# B&R Automation Studio project Lib1Lab1
Automation Studio 4.5.2.102

## Configuration Config1

CPU 4PP065.0571-P74, AutomationRuntime D4.52, Build 4.1.2, Vc V4.52.0

### Task classes (Cpu.sw)
```
Cyclic#1:
  Program <- Program.prg
Binaries: udbdef, TCData, ashwd, User, asfw, arconfig, sysconf, Role, ashwac, iomap
Libraries: LOR
```

### Hardware
```
4PP065_0571_P74 : 4PP065.0571-P74 v1.1.2.0
  Connector IF4:
    SubnetMask = 255.255.255.0
    InaNodeNumber = 1
  Connector IF5:
    ActivateDevice = 1
    Mode = Manual
    InternetAddress = 10.0.1.10
    SubnetMask = 255.255.255.0
  ConfigurationID = labBR
```

## Logical view

Binary libraries used (declarations not repeated): operator, runtime, astime, AsIecCon

### Package Logical/Libraries - Global libraries

### Library Logical/Libraries/LOR (ANSIC)

#### LOR.fun
```iecst
{REDUND_ERROR} FUNCTION_BLOCK FB_Integrator (*TODO: Add your comment here*) (*$GROUP=User,$CAT=User,$GROUPICON=User.png,$CATICON=User.png*)
	VAR_INPUT
		in : REAL;
	END_VAR
	VAR_OUTPUT
		out : REAL;
	END_VAR
	VAR
		dt : REAL;
	END_VAR
END_FUNCTION_BLOCK

{REDUND_ERROR} FUNCTION_BLOCK FB_Motor (*TODO: Add your comment here*) (*$GROUP=User,$CAT=User,$GROUPICON=User.png,$CATICON=User.png*)
	VAR_INPUT
		u : REAL;
	END_VAR
	VAR_OUTPUT
		phi : REAL;
		w : REAL;
	END_VAR
	VAR
		integrator : FB_Integrator;
		Tm : REAL;
		ke : REAL;
		dt : REAL;
	END_VAR
END_FUNCTION_BLOCK

{REDUND_ERROR} FUNCTION_BLOCK FB_Regulator (*TODO: Add your comment here*) (*$GROUP=User,$CAT=User,$GROUPICON=User.png,$CATICON=User.png*)
	VAR_INPUT
		e : REAL; (*рассогласование между задающим воздействием и реальной скоростью вращения вала ДПТ об/мин*)
	END_VAR
	VAR_OUTPUT
		u : REAL; (*напряжение на выходе ДПТ В*)
	END_VAR
	VAR
		k_p : REAL; (*П коэф регулятора*)
		k_i : REAL; (*И коэф регулятора*)
		integrator : FB_Integrator; (*Интегратор*)
		iyOld : REAL; (*храниение предыдущего значения схемы противонакопления*)
		max_abs_value : REAL; (*Umax*)
		dt : REAL; (*хе-хе-хе*)
		e_kp : REAL; (*промежуточное значение вычесления*)
	END_VAR
END_FUNCTION_BLOCK
```

#### FB_Integrator.c
```c
#include <bur/plctypes.h>
#ifdef __cplusplus
	extern "C"
	{
#endif
	#include "LOR.h"
#ifdef __cplusplus
	};
#endif
/* TODO: Add your comment here */
void FB_Integrator(struct FB_Integrator* inst)
{
	inst->out += inst->in;
}
```

#### FB_Motor.c
```c
#include <bur/plctypes.h>
#ifdef __cplusplus
	extern "C"
	{
#endif
	#include "LOR.h"
#ifdef __cplusplus
	};
#endif
/* TODO: Add your comment here */
void FB_Motor(struct FB_Motor* inst)
{
	inst->integrator.in = (inst->u/inst->ke - inst->w)*inst->dt/inst->Tm;
	inst->integrator.out = inst->w;
	FB_Integrator(&(inst->integrator));
	inst->integrator.in = inst->w * inst->dt;
	inst->integrator.out = inst->phi;
	FB_Integrator(&(inst->integrator));
	inst->phi = inst->integrator.out;
}
```

#### FB_Regulator.c
```c
#include <bur/plctypes.h>
#ifdef __cplusplus
	extern "C"
	{
#endif
	#include "LOR.h"
#ifdef __cplusplus
	};
#endif
/* TODO: Add your comment here */
void FB_Regulator(struct FB_Regulator* inst)
{
	inst->integrator.in=inst->e * inst->k_i * inst->dt + inst->iyOld;
	FB_Integrator(&(inst->integrator));
	inst->e_kp=inst->e*inst->k_p;
	inst->e_kp=(inst->e_kp > inst->max_abs_value || inst->e_kp < - inst->max_abs_value)?((inst->e_kp>0)?inst->max_abs_value:-inst->max_abs_value):inst->e_kp;
	inst->e_kp+=inst->integrator.out;
	inst->u=(inst->e_kp > inst->max_abs_value || inst->e_kp < - inst->max_abs_value)?((inst->e_kp>0)?inst->max_abs_value:-inst->max_abs_value):inst->e_kp;
	inst->iyOld=inst->u-inst->e_kp;
}
```

### Program Logical/Program (ANSIC)

#### Main.cpp - Init, cyclic, exit code
```cpp
#include <bur/plctypes.h>

#ifdef _DEFAULT_INCLUDES
	#include <AsDefault.h>
#endif

// amount of memory to be allocated for heap storage must be specified for every ANSI C++ program with the bur_heap_size variable
unsigned long bur_heap_size = 0xFFFF;

void _INIT ProgramInit(void)
{
	fb_motor.dt=0.0001;
	fb_motor.ke=2;
	fb_motor.Tm=0.4;
	fb_motor.integrator.dt=0.0001;

	fb_motor2.dt=0.0001;
	fb_motor2.ke=2;
	fb_motor2.Tm=0.4;
	fb_motor2.integrator.dt=0.0001;

	fb_regulator.dt=0.0001;
	fb_regulator.k_p=8;
	fb_regulator.k_i=20;
	fb_regulator.max_abs_value=24;
	fb_regulator.integrator.dt=0.0001;

	enable=1;
	count=0;

}

void _CYCLIC ProgramCyclic(void)
{
	if(enable)
	{
		count+=10;
		if(count<=2500)
		{
			speed=0;
		}

		else
		{
			speed=6;
			if(count>=5000)
			{
				count=0;
			}
		}
	}
	fb_regulator.e=speed - fb_motor.w;
	fb_motor2.u=speed;
	FB_Regulator(&fb_regulator);
	fb_motor.u=fb_regulator.u;
	FB_Motor(&fb_motor);
	FB_Motor(&fb_motor2);

}

void _EXIT ProgramExit(void)
{
	// Insert code here

}
```

#### Variables.var - Local variables
```iecst
VAR
	fb_regulator : FB_Regulator;
	fb_motor : FB_Motor;
	fb_motor2 : FB_Motor;
	speed : REAL;
	enable : BOOL;
	count : INT;
END_VAR
```

Listed in the project but not available here: Logical/Global.typ, Logical/Global.var, Logical/Program/Types.typ
